// TwinCAT 3 PLC project UtilitiesLibraryPractice
// ProgramVersion: 3.1.4024.0
// libraries:
//   LiquidFilling, * (InTimeTec)
//   Tc2_Standard, * (Beckhoff Automation GmbH)
//   Tc2_System, * (Beckhoff Automation GmbH)
//   Tc2_Utilities, * (Beckhoff Automation GmbH)
//   Tc3_Module, * (Beckhoff Automation GmbH)
// project tree:
//   DUTs/ E_EventType.TcDUT, ST_Event.TcDUT
//   / PlcTask.TcTTO
//   POUs/ FB_EventBuffer.TcPOU, FB_OpenFile.TcPOU, FB_ProfilerPractice.TcPOU, MAIN.TcPOU
//   POUs/TimerExample1/ FB_Factory.TcPOU
//   POUs/TimerExample2/ FB_LeakDetection.TcPOU
// (motion and I/O tree: see PLC project instructions_practice)
// real-time tasks:
//   TASK PlcTask: cycle T#10ms, priority 20, ADS port 350
//   TASK PlcTask1: cycle T#10ms, priority 22, ADS port 351
//   TASK PlcTask2: cycle T#10ms, priority 21, ADS port 352
//   TASK PlcTask3: cycle T#10ms, priority 23, ADS port 353
//   TASK PlcTask4: cycle T#10ms, priority 24, ADS port 354
//   TASK PlcTask5: cycle T#10ms, priority 25, ADS port 355

CONFIGURATION UtilitiesLibraryPractice
    RESOURCE PLC ON TwinCAT3
        TASK PlcTask(INTERVAL := T#10ms, PRIORITY := 25);
        PROGRAM MAIN WITH PlcTask : MAIN;
    END_RESOURCE
END_CONFIGURATION

// ---- DUTs/E_EventType.TcDUT
{attribute 'qualified_only'}
{attribute 'strict'}
TYPE E_EventType :
(
	Alarm := 0,
	Message := 1
);
END_TYPE

// ---- DUTs/ST_Event.TcDUT
TYPE ST_Event :
STRUCT
	eEventType : E_EventType;
	eEventSeverity : TcEventSeverity;
	nEventIdentity : UDINT;
	sEventText : STRING(255);
	dtTimestamp : DATE_AND_TIME;
END_STRUCT
END_TYPE

// ---- POUs/MAIN.TcPOU
PROGRAM MAIN
VAR
	stEvent : ST_Event;
	
	fbEventBuffer : FB_EventBuffer;
	fbTank : FB_StationController;
	fbFactory : FB_Factory;
	fbLeakDetection  : FB_LeakDetection;
	
	bAddEvent : BOOL;
	bRemoveEvent : BOOL;
	
	bAddEventError : BOOL;
	bGetRemoveEventError : BOOL;
	bGetEvent : ST_Event;
	bStart: BOOL;
	
	fbProfilerPractice : FB_ProfilerPractice;
	
	fbOpenFile : FB_OpenFile;
END_VAR

IF bAddEvent THEN
	fbEventBuffer.AddEvent(stEvent := stEvent, bError => bAddEventError);
	bAddEvent := FALSE;
END_IF

IF bRemoveEvent THEN
	fbEventBuffer.GetAndRemoveEvent(stEvent => bGetEvent, bError => bGetRemoveEventError);
	bRemoveEvent := FALSE;
END_IF
IF bStart THEN
	fbProfilerPractice();
END_IF

//fbOpenFile();
//fbFactory();
fbLeakDetection();

END_PROGRAM

// ---- POUs/FB_EventBuffer.TcPOU
FUNCTION_BLOCK FB_EventBuffer

VAR
	fbBuffer : FB_MemRingBuffer;
	aEventArray : ARRAY[0..MAX_EVENTS_TO_BE_STORED] OF BYTE ;
END_VAR
VAR CONSTANT
	MAX_NUMBER_OF_EVENTS : INT := 5;
	SIZE_OF_EVENT : UDINT := SIZEOF(ST_Event);
	MAX_EVENTS_TO_BE_STORED : UDINT := SIZE_OF_EVENT * MAX_NUMBER_OF_EVENTS;
END_VAR

METHOD AddEvent
VAR_INPUT
	stEvent : ST_Event;
END_VAR
VAR_OUTPUT
	bError : BOOL;
END_VAR
fbBuffer.A_AddTail(
					pWrite := ADR(stEvent),
					cbWrite := SIZEOF(stEvent),
					pBuffer := ADR(aEventArray),
					cbBuffer := SIZEOF(aEventArray)
					);
bError := NOT fbBuffer.bOk;
END_METHOD

METHOD GetAndRemoveEvent
VAR_OUTPUT
	stEvent: ST_Event;
	bError: BOOL;
END_VAR
fbBuffer.A_RemoveHead(
					pRead := ADR(stEvent),
					cbRead := SIZEOF(stEvent),
					pBuffer := ADR(aEventArray),
					cbBuffer := SIZEOF(aEventArray)
					);
bError := NOT fbBuffer.bOk;
END_METHOD

END_FUNCTION_BLOCK

// ---- POUs/TimerExample1/FB_Factory.TcPOU
FUNCTION_BLOCK FB_Factory

VAR
	fbTon : TON;
	fbTof : TOF;
	
	bMotorOn : BOOL;
	bFanOn : BOOL;
	
	tFanStartDelay : TIME := T#3S;
	tFanOffDelay : TIME := T#10s;
END_VAR


	fbTon(IN := bMotorOn, PT := tFanStartDelay);
	IF fbTon.Q THEN
		bFanOn := TRUE;
	END_IF
	fbTof(IN := bMotorOn , PT := tFanOffDelay);
	IF NOT fbTof.Q THEN
		bFanOn := FALSE;
	END_IF

END_FUNCTION_BLOCK

// ---- POUs/TimerExample2/FB_LeakDetection.TcPOU
FUNCTION_BLOCK FB_LeakDetection

VAR
	bValveOpen : BOOL;
	bFlowSensor : BOOL;
	
	fbTon : TON;
	fbTp : TP;
	
	bAlarm : BOOL;
	tFlowTime : TIME := T#2S;
	tAlarmDuration : TIME := T#5S;
END_VAR

fbTon(IN := bValveOpen , PT := tFlowTime);
IF fbTon.Q THEN
	bFlowSensor := TRUE;
ELSE
	bFlowSensor := FALSE;
END_IF

fbTp(IN := bFlowSensor,PT := tAlarmDuration);
bAlarm := fbTp.Q;

END_FUNCTION_BLOCK

// ---- POUs/FB_ProfilerPractice.TcPOU
FUNCTION_BLOCK FB_ProfilerPractice

VAR
	fbProfiler : PROFILER;
	stProfilerResult : PROFILERSTRUCT;
	nFactorial : ULINT;
	n : ULINT := 1000;
END_VAR

fbProfiler(START := TRUE, RESET := FALSE);
Factorial(n := n , nFactorialValue => nFactorial );
fbProfiler(START := FALSE);
stProfilerResult := fbProfiler.DATA;

METHOD Factorial
VAR_INPUT
	n : ULINT;
END_VAR
VAR
	nCounter : ULINT;
END_VAR
VAR_OUTPUT
	nFactorialValue : ULINT := 1;
END_VAR
FOR nCounter := 1 TO n DO
	nFactorialValue := nFactorialValue * nCounter;
END_FOR
END_METHOD

END_FUNCTION_BLOCK

// ---- POUs/FB_OpenFile.TcPOU
FUNCTION_BLOCK FB_OpenFile

VAR
	fbStartProcess : NT_StartProcess := (NETID := '',TMOUT := T#5S );
	bError : BOOL;
END_VAR

fbStartProcess(PATHSTR := 'C:\Windows\notepad.exe',
				DIRNAME := 'D:\Temp\',
				COMNDLINE := 'Event.txt',
				START := TRUE
				);
bError := fbStartProcess.ERR;

END_FUNCTION_BLOCK
